FUNCTION_BLOCK FlushDone (* Basic Function Block Type *)
  (* Standard: 61499-2 *)
  (* Version 0.0, 6/20/2026, Schneider Electric, Template *)
  PACKAGE SE.Nereda;
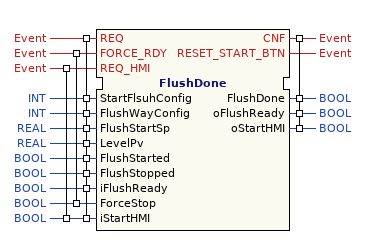
  EVENT_INPUT
    REQ WITH StartFlsuhConfig, FlushStartSp, LevelPv, FlushWayConfig, FlushStarted, FlushStopped, iFlushReady, iStartHMI; (* Normal Execution Request *)
    FORCE_RDY WITH ForceStop;
    REQ_HMI WITH iStartHMI;
  END_EVENT
  EVENT_OUTPUT
    CNF WITH FlushDone, oFlushReady, oStartHMI; (* Execution Confirmation *)
    RESET_START_BTN;
  END_EVENT
  VAR_INPUT
    StartFlsuhConfig : INT; (* Input event qualifier *)
    FlushWayConfig : INT;
    FlushStartSp : REAL;
    LevelPv : REAL;
    FlushStarted : BOOL;
    FlushStopped : BOOL;
    iFlushReady : BOOL;
    ForceStop : BOOL;
    iStartHMI : BOOL;
  END_VAR
  VAR_OUTPUT
    FlushDone : BOOL; (* Output event qualifier *)
    oFlushReady : BOOL;
    oStartHMI : BOOL;
  END_VAR
  VAR
    FirstFlush : BOOL;
  END_VAR
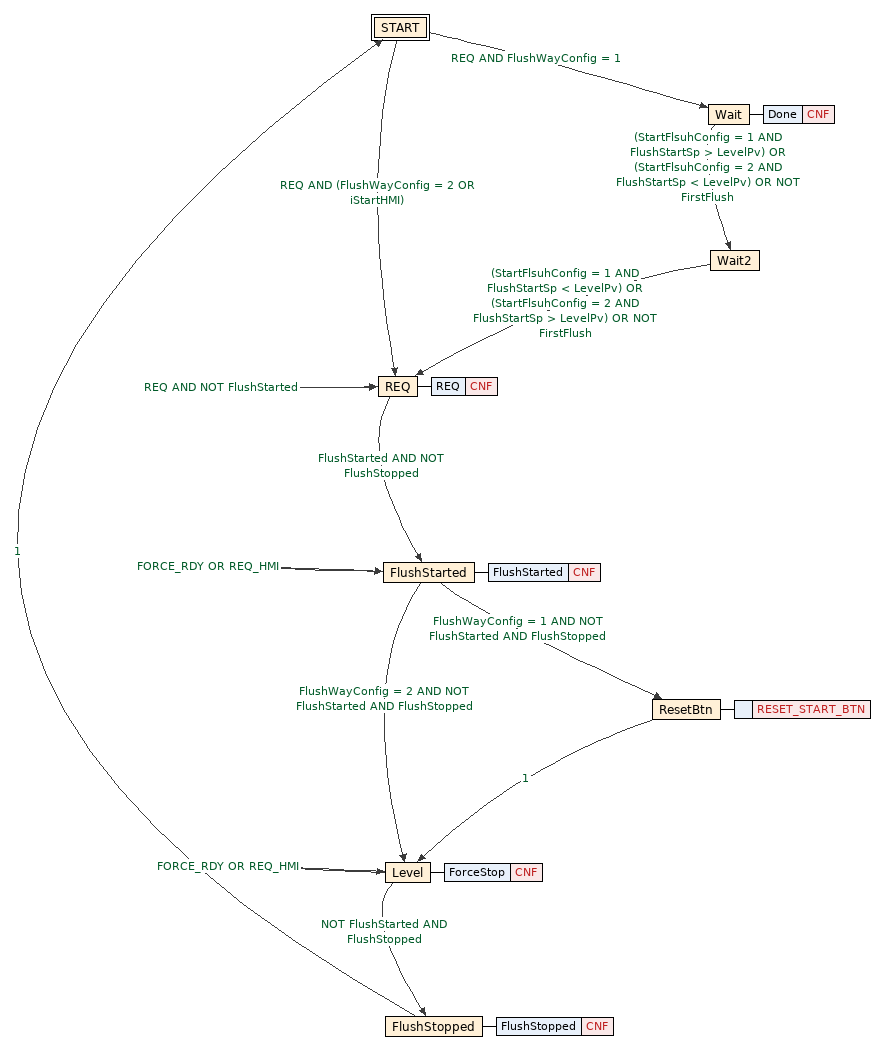
  EC_STATES
    START; (* Initial State *)
    REQ : REQ -> CNF;
    FlushStarted : FlushStarted -> CNF;
    Level : ForceStop -> CNF;
    FlushStopped : FlushStopped -> CNF;
    ResetBtn : -> RESET_START_BTN;
    Wait : Done -> CNF;
    Wait2;
  END_STATES
  EC_TRANSITIONS
    START TO Wait := REQ AND FlushWayConfig = 1;
    REQ TO REQ := REQ AND NOT FlushStarted;
    REQ TO FlushStarted := FlushStarted AND NOT FlushStopped;
    FlushStarted TO Level := FlushWayConfig = 2 AND NOT FlushStarted AND FlushStopped;
    Level TO FlushStopped := NOT FlushStarted AND FlushStopped;
    FlushStopped TO START := 1;
    FlushStarted TO FlushStarted := FORCE_RDY OR REQ_HMI;
    Level TO Level := FORCE_RDY OR REQ_HMI;
    FlushStarted TO ResetBtn := FlushWayConfig = 1 AND NOT FlushStarted AND FlushStopped;
    ResetBtn TO Level := 1;
    START TO REQ := REQ AND (FlushWayConfig = 2 OR iStartHMI);
    Wait TO Wait2 := (StartFlsuhConfig = 1 AND FlushStartSp > LevelPv) OR (StartFlsuhConfig = 2 AND FlushStartSp < LevelPv) OR NOT FirstFlush;
    Wait2 TO REQ := (StartFlsuhConfig = 1 AND FlushStartSp < LevelPv) OR (StartFlsuhConfig = 2 AND FlushStartSp > LevelPv) OR NOT FirstFlush;
  END_TRANSITIONS
  ALGORITHM REQ IN ST: (* Normally executed algorithm *)
;
// StartFlsuhConfig = 1 => Flush SP <= PV
// StartFlsuhConfig = 2 => Flush SP >= PV
// FlushWayConfig = 1 => Flush Once
// FlushWayConfig = 2 => Cyclic Flush

IF iFlushReady THEN
	IF FlushWayConfig = 1 THEN
		IF StartFlsuhConfig = 1 THEN
			IF FlushStartSp <= LevelPv THEN
				FlushDone := FALSE;
				oFlushReady := TRUE;
			ELSE
				FlushDone := TRUE;
			END_IF;
		ELSIF StartFlsuhConfig = 2 THEN
			IF FlushStartSp >= LevelPv THEN
				FlushDone := FALSE;
				oFlushReady := TRUE;
			ELSE
				FlushDone := TRUE;
			END_IF;
		END_IF;

	ELSIF FlushWayConfig = 2 THEN
		oFlushReady := TRUE;
		FlushDone := TRUE;
	END_IF;
ELSE
	FlushDone := TRUE;
	oFlushReady := iFlushReady;
END_IF;

// StartFlsuhConfig = 1 => Flush SP <= PV
// StartFlsuhConfig = 2 => Flush SP >= PV
// FlushWayConfig = 1 => Flush Once
// FlushWayConfig = 2 => Cyclic Flush

IF iStartHMI THEN
	oStartHMI := iStartHMI;
	IF FlushWayConfig = 1 THEN
		IF StartFlsuhConfig = 1 THEN
			FlushDone := FALSE;
			oFlushReady := TRUE;
		ELSIF StartFlsuhConfig = 2 THEN
			FlushDone := FALSE;
			oFlushReady := TRUE;
		END_IF;

	ELSIF FlushWayConfig = 2 THEN
		oFlushReady := TRUE;
		FlushDone := TRUE;
	END_IF;
END_IF;
  END_ALGORITHM
  ALGORITHM FlushStarted IN ST:
;
FirstFlush := TRUE;
IF NOT ForceStop THEN
	IF FlushWayConfig = 1 THEN
		FlushDone := TRUE;
		oFlushReady := TRUE;
	ELSIF FlushWayConfig = 2 THEN
		FlushDone := FALSE;
		oFlushReady := iFlushReady;
	END_IF;
ELSE
	oFlushReady := iFlushReady;
END_IF;
  END_ALGORITHM
  ALGORITHM FlushStopped IN ST:
;
IF FlushWayConfig = 1 THEN
	FlushDone := TRUE;
	oFlushReady := FALSE;
ELSIF FlushWayConfig = 2 THEN
	FlushDone := FALSE;
	oFlushReady := iFlushReady;
END_IF;
  END_ALGORITHM
  ALGORITHM ForceStop IN ST:
;
IF ForceStop THEN
	oFlushReady := iFlushReady;
END_IF;
  END_ALGORITHM
  ALGORITHM Done IN ST:
;
FlushDone := TRUE;
oFlushReady := FALSE;
  END_ALGORITHM
END_FUNCTION_BLOCK
